// TIA Portal V20 export
DATA_BLOCK "iDB_Valve_Inlet"   // DB900
// EXAMPLE instance DB for FB_Valve - one valve, wired in examples/calling-network.ir. START VALUES ARE DOWNLOAD-TIME ONLY and every command member is overwritten by the caller each scan, so the values that actually matter here are the two SETTINGS: FTTime, which must cover this actuator's travel in its slower direction, and EnableUPSTime. Both ship non-zero on purpose - a zero fail-to time raises both faults during every legitimate transit. The whole struct is RETAIN, which is what C-132 makes possible and what keeps a latched fault alive across a power cycle; note that this retains the entire interface, not only the latched causes.
// stored: InstanceOfName FB_Valve, InstanceOfType FB
"FB_Valve"
   // VAR RETAIN
   //    IO { S7_SetPoint := 'True'} : "UDT_Valve";
   // END_VAR
   // VAR
   //    FBOpen : Bool := FALSE;
   //    CycleEdge : Bool := FALSE;
   //    CyclePrev : Bool := FALSE;
   //    FTTimeMS : DInt := 0;
   //    EnableUPSTimeMS : DInt := 0;
   //    FailToOpenTimer { S7_SetPoint := 'True'} : TON_TIME;
   //    FailToCloseTimer { S7_SetPoint := 'True'} : TON_TIME;
   //    EnableUpstreamTimer { S7_SetPoint := 'True'} : TON_TIME;
   //    CycleDebounceTimer { S7_SetPoint := 'True'} : TON_TIME;
   // END_VAR
BEGIN
   IO.InHand := FALSE;
   IO.AutoOpenSignal := FALSE;
   IO.HandOpenSignal := FALSE;
   IO.PositionFB := FALSE;
   IO.PositionValid := FALSE;
   IO.FBSenseInvert := FALSE;
   IO.FaultFB := FALSE;
   IO.SystemHealthy := FALSE;
   IO.InhibitValve := FALSE;
   IO.FaultReset := FALSE;
   IO.FTTime := 10.0;
   IO.EnableUPSTime := 2.0;
   IO.FailCloseCritical := FALSE;
   IO.SuppFTO := FALSE;
   IO.SuppFTC := FALSE;
   IO.OpenValve := FALSE;
   IO.UPSEnable := FALSE;
   IO.FTO := FALSE;
   IO.FTC := FALSE;
   IO.ExtFault := FALSE;
   IO.OverrideActive := FALSE;
   IO.FaultActive := FALSE;
   IO.CriticalActive := FALSE;
   IO.ErrorActive := FALSE;
   IO.CycleCount := 0;
   IO.Telemetry := 0;
   IO.Alarm := 16#0;
   IO.SuppCause := 0;
   FailToOpenTimer.PT := T#0MS;
   FailToOpenTimer.ET := T#0MS;
   FailToOpenTimer.IN := FALSE;
   FailToOpenTimer.Q := FALSE;
   FailToCloseTimer.PT := T#0MS;
   FailToCloseTimer.ET := T#0MS;
   FailToCloseTimer.IN := FALSE;
   FailToCloseTimer.Q := FALSE;
   EnableUpstreamTimer.PT := T#0MS;
   EnableUpstreamTimer.ET := T#0MS;
   EnableUpstreamTimer.IN := FALSE;
   EnableUpstreamTimer.Q := FALSE;
   CycleDebounceTimer.PT := T#0MS;
   CycleDebounceTimer.ET := T#0MS;
   CycleDebounceTimer.IN := FALSE;
   CycleDebounceTimer.Q := FALSE;
END_DATA_BLOCK
